(********************* G.D S.p.A. - Technical Department ***********************************
This program has been generated automatically from Application Designer DE&F
********************************************************************************************)
PROGRAM dbg_csp_transfer_main_safety_drives_commonconfiguration
VAR
  rack_smes_sis_shd : safety_integrated_series_shadow;
  standalone_smes_sis_shd : safety_integrated_series_shadow;
END_VAR

_objects_manager();

IF	g_application_status <> APPLICATION_STATUS_RUNNING
THEN
	RETURN;
END_IF

CASE process_get_mode(CONVERSION_this := dbg_root.prc) OF
	MODE_ABSENT,
	MODE_INACTIVE:
		RETURN;
	MODE_TEST:
		RETURN;
END_CASE

ACTION _objects_manager:
IF	objects_initialization()
THEN
	safety_integrated_series_shadow_init(
		sim_mode:= SHADOW_SIMULATION_MODE_AUTOMATIC, 
		father:= csp_transfer_main_safety_drives_commonconfiguration.rack_smes_sis, 
		process:= dbg_root.prc, 
		CONVERSION_this:= rack_smes_sis_shd);

	safety_integrated_series_shadow_init(
		sim_mode:= SHADOW_SIMULATION_MODE_AUTOMATIC, 
		father:= csp_transfer_main_safety_drives_commonconfiguration.standalone_smes_sis, 
		process:= dbg_root.prc, 
		CONVERSION_this:= standalone_smes_sis_shd);

	RETURN;
END_IF

IF	objects_running()
THEN
	safety_integrated_series_shadow_cycle(rack_smes_sis_shd);
	safety_integrated_series_shadow_cycle(standalone_smes_sis_shd);
END_IF
END_ACTION

END_PROGRAM

(* stored: Version 1.1.0.1, ProductVersion 3.1.4022.12
   POU dbg_csp_transfer_main_safety_drives_commonconfiguration: Id {d03ec8dc-93e2-4c11-9cf5-8d4d2e80da3c}, SpecialFunc None
   Action _objects_manager: Id {9589c5a5-85c6-4f42-99b1-bfa90566e5da} *)
